TYPE IOExpantionMessage_t :
STRUCT
	{warning 'define variables'}
END_STRUCT
END_TYPE

(* stored: Version 1.1.0.1
   DUT IOExpantionMessage_t: Id {66fa93d8-0733-47de-88e3-df9986d138db} *)
